PROGRAM INTERNAL P_Enumerator_Example
VAR
	bStart : BOOL;
	sValue : STRING(255);
	dtTime : DT :=  DT#2023-5-8-12:55:23;
	fbString_Builder1,
	fbString_Builder2 : FB_String_Builder;
	ipEnumerator : I_Enumerator;
END_VAR

IF bStart THEN
	bStart := FALSE;
	
	fbString_Builder1
		.Clear()
		.Append('   I love cats.')
		.Append('The time is: ').Append_Any(dtTime).Append('.')
		.Trim_Whitespace(T_Whitespace_Location.Both);
	
	ipEnumerator := fbString_Builder1.Get_Enumerator();
	WHILE ipEnumerator.Next() DO
		fbString_Builder2.Append(ipEnumerator._Current);
		END_WHILE
		
	sValue := fbString_Builder2.Get_String();
	END_IF

END_PROGRAM

(* stored: Version 1.1.0.1, ProductVersion 3.1.4024.4
   POU P_Enumerator_Example: Id {b227b542-53a7-4513-abcd-f9f25dca4fa9}, SpecialFunc None *)
